(* CoDeSys 2.3.9.22 project: pr4.pro *)
(* Libraries: Util.lib 18.5.10 15:14:28, STANDARD.LIB 4.10.05 11:14:46, IECSFC.LIB 13.4.06 15:51:28, ANALYZATION.LIB 5.10.99 09:05:06 *)

(* PLC configuration (modules and I/O channels)
PLC 150 I [Root] node -1, in %IB0 out %QB0 {MinCycleLength = 1; MaxCycleLength = 5000}
  Discrete input 6 bit [ID100] node 0, in %IB0 out %QB0 {Filtrationtime = 10; Filtrationtime = 10; Filtrationtime = 10; Filtrationtime = 10; Filtrationtime = 10; Filtrationtime = 10; Visibility = No; PinCount = 6; WatchDogPeriod = 1000; PollPeriod = 1}
    AT %IX0.0 [BitInput]
    AT %IX0.1 [BitInput]
    AT %IX0.2 [BitInput]
    AT %IX0.3 [BitInput]
    AT %IX0.4 [BitInput]
    AT %IX0.5 [BitInput]
  Discrete output 4 bit [ID101] node 1, in %IB1 out %QB1 {PinCount = 4; SafeValueBool = FALSE; SafeValueBool = FALSE; SafeValueBool = FALSE; SafeValueBool = FALSE; Visibility = No}
    AT %QX1.0 [BitOutput]
    AT %QX1.1 [BitOutput]
    AT %QX1.2 [BitOutput]
    AT %QX1.3 [BitOutput]
  Special output [ID104] node 2, in %IB2 out %QB2 {Visibility = No; PinCount = 1}
    AT %QX2.0 [BitOutput] Special output
  Unifed signal sensor [ID700] node 3, in %IB3 out %QB3 {Type_of_sensor700 = IT_0_20; measure_interval = 0.8; ainlow = 0; ainhigh = 20; first_cor_point = 0; first_delta = 0; second_cor_point = 0; second_delta = 0; third_cor_point = 0; third_delta = 0; Visibility = No}
    AT %ID3.0 [FloatInput] Value
    AT %IW3.1 [WordInput] Circular time
    Analog Input [ID107] node 0, in %IB3.0 out %QB3.0
  Unifed signal sensor [ID700] node 4, in %IB4 out %QB4 {Type_of_sensor700 = IT_0_20; measure_interval = 0.8; ainlow = 0; ainhigh = 20; first_cor_point = 0; first_delta = 0; second_cor_point = 0; second_delta = 0; third_cor_point = 0; third_delta = 0; Visibility = No}
    AT %ID4.0 [FloatInput] Value
    AT %IW4.1 [WordInput] Circular time
    Analog Input [ID107] node 0, in %IB4.0 out %QB4.0
  Unifed signal sensor [ID700] node 5, in %IB5 out %QB5 {Type_of_sensor700 = IT_0_20; measure_interval = 0.8; ainlow = 0; ainhigh = 20; first_cor_point = 0; first_delta = 0; second_cor_point = 0; second_delta = 0; third_cor_point = 0; third_delta = 0; Visibility = No}
    AT %ID5.0 [FloatInput] Value
    AT %IW5.1 [WordInput] Circular time
    Analog Input [ID107] node 0, in %IB5.0 out %QB5.0
  Unifed signal sensor [ID700] node 6, in %IB6 out %QB6 {Type_of_sensor700 = IT_0_20; measure_interval = 0.8; ainlow = 0; ainhigh = 20; first_cor_point = 0; first_delta = 0; second_cor_point = 0; second_delta = 0; third_cor_point = 0; third_delta = 0; Visibility = No}
    AT %ID6.0 [FloatInput] Value
    AT %IW6.1 [WordInput] Circular time
    Analog Input [ID107] node 0, in %IB6.0 out %QB6.0
  Analog output [ID106] node 7, in %IB7 out %QB7 {DAC_Type = Current 4-20mA; Analog_offset_correction = 0; Analog_full_range_correction = 0; SafeValueFloat = 0; Visibility = No}
    AT %QD7.0 [FloatOutput] Value
  Analog output [ID106] node 8, in %IB8 out %QB8 {DAC_Type = Current 4-20mA; Analog_offset_correction = 0; Analog_full_range_correction = 0; SafeValueFloat = 0; Visibility = No}
    AT %QD8.0 [FloatOutput] Value
*)

(* POU PLC_PRG, CFC *)
PROGRAM PLC_PRG
VAR
	start: BOOL;
	pipe: BOOL;
	ctu1: CTU;
	blink1: BLINK;
	ctu2: CTU;
	wagon: REAL;
	rs1: RS;
	givePipe: BOOL;
	pipeVanish: BOOL;
	rs2: RS;
	givePipeC1: BOOL;
	givePipeC2: BOOL;
	pipeVanishC1: BOOL;
	pipeVanishC2: BOOL;
	rs3: RS;
	ctu3: CTU;
	ctu4: CTU;
	pipe1Y: REAL;
	pipe2Y: REAL;
	pipe2X: REAL;
	ctu5: CTU;
	pipe1X: REAL;
	stop: BOOL;
	loadEnd: BOOL;
	blink2: BLINK;
	wagon1: REAL;
	C1: BOOL;
	C2: BOOL;
	ctu6: CTU;
	rs4: RS;
	ctu7: CTU;
	givePipeC1ON: BOOL;
	P9: BOOL;
	ctu8: CTU;
	removePipeC1: BOOL;
	removePipeC2: BOOL;
	rs5: RS;
	ctu9: CTU;
	givePipeC2ON: BOOL;
	P0: BOOL;
	P5: BOOL;
	P6: BOOL;
	P4: BOOL;
	P3: BOOL;
	P1: BOOL;
	P2: BOOL;
	P8: BOOL;
END_VAR
VAR (* helpers for the ST form of the networks *)
	_t369 : BOOL;
	_t164 : BOOL;
	_t287 : BOOL;
	_t446 : BOOL;
	_t193 : BOOL;
	_t190 : REAL;
	_t207 : REAL;
	_t237 : REAL;
	_t321 : REAL;
	_t357 : REAL;
	_t214 : BOOL;
	_t430 : BOOL;
	_t250 : REAL;
	_t294 : REAL;
	_t315 : BOOL;
	_t445 : BOOL;
	_t241 : BOOL;
	_t231 : REAL;
	_t345 : REAL;
	_t431 : BOOL;
	_t350 : BOOL;
	_t427 : BOOL;
	_t440 : BOOL;
END_VAR
_CFC_ (* Continuous Function Chart, elements in execution order *)
#0 AND(#7.Q1, NOT #8.Q)
#1 AND(NOT stop, #16.OUT)
#2 AND(#1, #35)
#3 loadEnd <= #2
#4 AND(#7.Q1, NOT #43.Q1)
#5 S pipeVanishC1 <= NOT givePipeC1
#6 R pipeVanishC1 <= #8.Q
#7 rs2:RS(SET: givePipeC1, RESET1: #58.Q)
#8 ctu1:CTU(CU: #25, RESET: #58.Q, PV: 14)
#9 AND(#7.Q1, #1, #4)
#10 ADD(#18, #42, #51, #59, #70)
#11 wagon <= #10
#12 AND(#1, #7.Q1, NOT #27.Q)
#13 C1 <= #12
#14 AND(#24, start)
#15 rs1:RS(SET: #14, RESET1: #58.Q)
#16 blink1:BLINK(ENABLE: #15.Q1, TIMELOW: T#0.1s, TIMEHIGH: T#0.1s)
#17 WORD_TO_REAL(#8.CV)
#18 MUL(#17, -1)
#19 EQ(wagon, 0)
#20 P9 <= #19
#21 AND(#7.Q1, NOT #27.Q)
#22 givePipeC1ON <= #21
#23 EQ(pipe1Y, -44)
#24 OR(#7.Q1, #43.Q1)
#25 AND(#9, NOT #8.Q)
#26 AND(#8.Q, #9, NOT #27.Q)
#27 ctu2:CTU(CU: #26, RESET: #58.Q, PV: 22)
#28 pipe1Y <= #40
#29 AND(#39.Q, #9, NOT #30.Q)
#30 ctu6:CTU(CU: #29, RESET: #58.Q, PV: 22)
#31 MUL(#55, -1)
#32 rs4:RS(SET: #33, RESET1: #58.Q)
#33 AND(removePipeC1, #30.Q)
#34 AND(#43.Q1, #1, #74)
#35 OR(#27.Q, #45.Q)
#36 WORD_TO_REAL(#27.CV)
#37 MUL(#36, -1)
#38 AND(#27.Q, #9, NOT #39.Q)
#39 ctu3:CTU(CU: #38, RESET: #58.Q, PV: 38)
#40 ADD(#37, #47, #31, #64)
#41 WORD_TO_REAL(#39.CV)
#42 MUL(#41, -1)
#43 rs3:RS(SET: givePipeC2, RESET1: #69.Q)
#44 AND(#34, NOT #45.Q)
#45 ctu4:CTU(CU: #44, RESET: #69.Q, PV: 22)
#46 WORD_TO_REAL(#45.CV)
#47 MUL(#46, -1)
#48 AND(#45.Q, #34, NOT #49.Q)
#49 ctu5:CTU(CU: #48, RESET: #69.Q, PV: 40)
#50 WORD_TO_REAL(#49.CV)
#51 MUL(#50, -1)
#52 R pipeVanishC1 <= #43.Q1
#53 AND(#1, #43.Q1, NOT #45.Q)
#54 C2 <= #53
#55 WORD_TO_REAL(#30.CV)
#56 S pipeVanishC1 <= #32.Q1
#57 AND(#32.Q1, #9, NOT #58.Q)
#58 ctu7:CTU(CU: #57, RESET: #58.Q, PV: 52)
#59 WORD_TO_REAL(#58.CV)
#60 AND(#34, NOT #61.Q, #49.Q)
#61 ctu8:CTU(CU: #60, RESET: #69.Q, PV: 22)
#62 P1 <= #90
#63 WORD_TO_REAL(#61.CV)
#64 MUL(#63, -1)
#65 rs5:RS(SET: #66, RESET1: #69.Q)
#66 AND(removePipeC2, #61.Q)
#67 S pipeVanishC1 <= #65.Q1
#68 AND(#65.Q1, #34, NOT #69.Q)
#69 ctu9:CTU(CU: #68, RESET: #69.Q, PV: 40)
#70 WORD_TO_REAL(#69.CV)
#71 S pipeVanishC2 <= #8.Q
#72 S pipeVanishC2 <= NOT givePipeC1
#73 R pipeVanishC2 <= #0
#74 AND(#43.Q1, NOT #7.Q1)
#75 AND(#43.Q1, NOT #45.Q)
#76 givePipeC2ON <= #75
#77 EQ(wagon, -52)
#78 P0 <= #77
#79 EQ(wagon, -40)
#80 P0 <= #79
#81 EQ(wagon, -52)
#82 P5 <= #81
#83 EQ(wagon, -40)
#84 P6 <= #83
#85 EQ(pipe1Y, 0)
#86 P3 <= #91
#87 EQ(pipe1Y, 0)
#88 AND(#87, givePipeC2ON)
#89 P4 <= #88
#90 AND(#81, #23)
#91 AND(#85, givePipeC1ON)
#92 EQ(pipe1Y, -44)
#93 P2 <= #94
#94 AND(#83, #92)
#95 EQ(wagon, -14)
#96 P8 <= #95
_END_CFC_
(* the same logic as Structured Text *)
_t369 := rs2.Q1 AND NOT ctu1.Q;
_t164 := NOT stop AND blink1.OUT;
loadEnd := _t164 AND _t287;
_t446 := rs2.Q1 AND NOT rs3.Q1;
IF NOT givePipeC1 THEN pipeVanishC1 := TRUE; END_IF;
IF ctu1.Q THEN pipeVanishC1 := FALSE; END_IF;
rs2(SET := givePipeC1, RESET1 := ctu7.Q);
ctu1(CU := _t193, RESET := ctu7.Q, PV := 14);
wagon := _t190 + _t207 + _t237 + _t321 + _t357;
C1 := _t164 AND rs2.Q1 AND NOT ctu2.Q;
rs1(SET := _t214 AND start, RESET1 := ctu7.Q);
blink1(ENABLE := rs1.Q1, TIMELOW := T#0.1s, TIMEHIGH := T#0.1s);
_t190 := WORD_TO_REAL(ctu1.CV) * (-1);
P9 := wagon = 0;
givePipeC1ON := rs2.Q1 AND NOT ctu2.Q;
_t430 := pipe1Y = (-44);
_t214 := rs2.Q1 OR rs3.Q1;
_t193 := (rs2.Q1 AND _t164 AND _t446) AND NOT ctu1.Q;
ctu2(CU := ctu1.Q AND (rs2.Q1 AND _t164 AND _t446) AND NOT ctu2.Q, RESET := ctu7.Q, PV := 22);
pipe1Y := _t250;
ctu6(CU := ctu3.Q AND (rs2.Q1 AND _t164 AND _t446) AND NOT ctu6.Q, RESET := ctu7.Q, PV := 22);
rs4(SET := _t315, RESET1 := ctu7.Q);
_t315 := removePipeC1 AND ctu6.Q;
_t241 := rs3.Q1 AND _t164 AND _t445;
_t287 := ctu2.Q OR ctu4.Q;
ctu3(CU := ctu2.Q AND (rs2.Q1 AND _t164 AND _t446) AND NOT ctu3.Q, RESET := ctu7.Q, PV := 38);
_t250 := (WORD_TO_REAL(ctu2.CV) * (-1)) + _t231 + (_t294 * (-1)) + _t345;
_t207 := WORD_TO_REAL(ctu3.CV) * (-1);
rs3(SET := givePipeC2, RESET1 := ctu9.Q);
ctu4(CU := _t241 AND NOT ctu4.Q, RESET := ctu9.Q, PV := 22);
_t231 := WORD_TO_REAL(ctu4.CV) * (-1);
ctu5(CU := ctu4.Q AND _t241 AND NOT ctu5.Q, RESET := ctu9.Q, PV := 40);
_t237 := WORD_TO_REAL(ctu5.CV) * (-1);
IF rs3.Q1 THEN pipeVanishC1 := FALSE; END_IF;
C2 := _t164 AND rs3.Q1 AND NOT ctu4.Q;
_t294 := WORD_TO_REAL(ctu6.CV);
IF rs4.Q1 THEN pipeVanishC1 := TRUE; END_IF;
ctu7(CU := rs4.Q1 AND (rs2.Q1 AND _t164 AND _t446) AND NOT ctu7.Q, RESET := ctu7.Q, PV := 52);
_t321 := WORD_TO_REAL(ctu7.CV);
ctu8(CU := _t241 AND NOT ctu8.Q AND ctu5.Q, RESET := ctu9.Q, PV := 22);
P1 := _t431;
_t345 := WORD_TO_REAL(ctu8.CV) * (-1);
rs5(SET := _t350, RESET1 := ctu9.Q);
_t350 := removePipeC2 AND ctu8.Q;
IF rs5.Q1 THEN pipeVanishC1 := TRUE; END_IF;
ctu9(CU := rs5.Q1 AND _t241 AND NOT ctu9.Q, RESET := ctu9.Q, PV := 40);
_t357 := WORD_TO_REAL(ctu9.CV);
IF ctu1.Q THEN pipeVanishC2 := TRUE; END_IF;
IF NOT givePipeC1 THEN pipeVanishC2 := TRUE; END_IF;
IF _t369 THEN pipeVanishC2 := FALSE; END_IF;
_t445 := rs3.Q1 AND NOT rs2.Q1;
givePipeC2ON := rs3.Q1 AND NOT ctu4.Q;
P0 := wagon = (-52);
P0 := wagon = (-40);
P5 := wagon = (-52);
P6 := wagon = (-40);
P3 := _t427;
P4 := (pipe1Y = 0) AND givePipeC2ON;
_t431 := (wagon = (-52)) AND _t430;
_t427 := (pipe1Y = 0) AND givePipeC1ON;
P2 := _t440;
_t440 := (wagon = (-40)) AND (pipe1Y = (-44));
P8 := wagon = (-14);
END_PROGRAM

(* Visualisation viz1
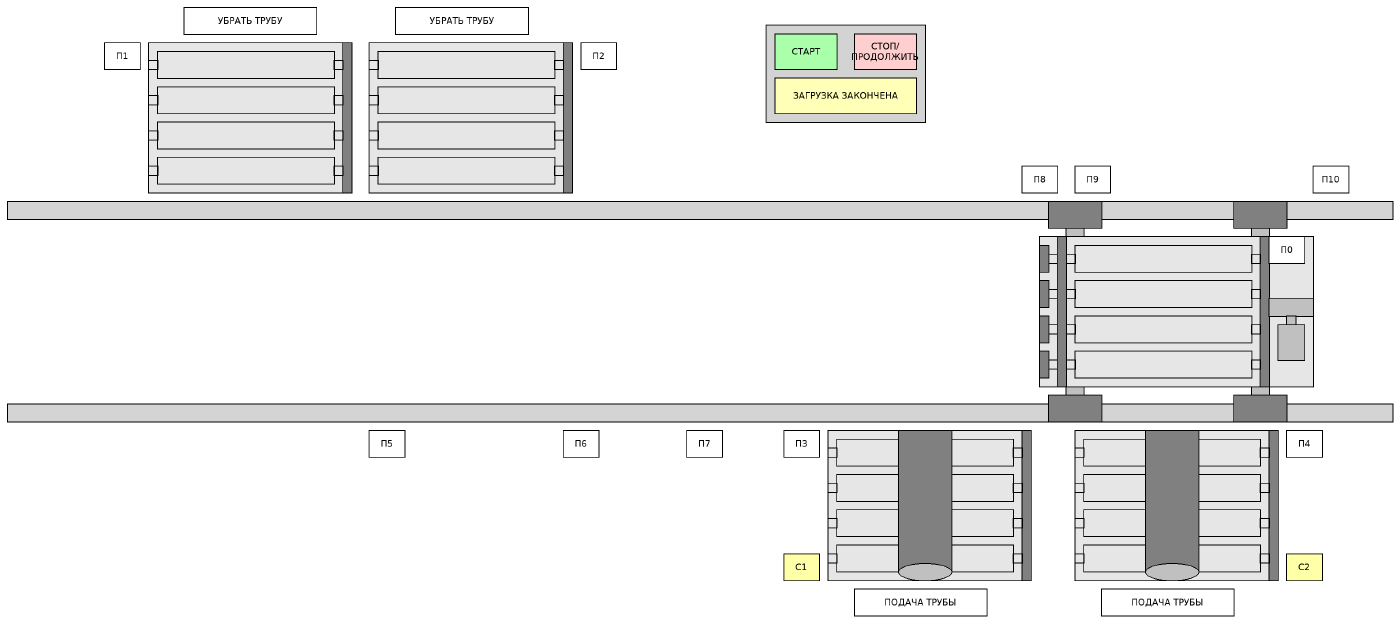
rectangle at (120,50)-(161,81): text "П1"; alarm colour if PLC_PRG.P1
rectangle at (660,50)-(701,81): text "П2"; alarm colour if PLC_PRG.P2
rectangle at (420,490)-(461,521): text "П5"; alarm colour if PLC_PRG.P5
rectangle at (640,490)-(681,521): text "П6"; alarm colour if PLC_PRG.P6
rectangle at (890,490)-(931,521): text "П3"; alarm colour if PLC_PRG.P3
rectangle at (780,490)-(821,521): text "П7"
rectangle at (1460,490)-(1501,521): text "П4"; alarm colour if PLC_PRG.P4
rectangle at (890,630)-(931,661): text "С1"; alarm colour if PLC_PRG.C1
rectangle at (1160,190)-(1201,221): text "П8"; alarm colour if PLC_PRG.P8
rectangle at (1220,190)-(1261,221): text "П9"; alarm colour if PLC_PRG.P9
rectangle at (1490,190)-(1531,221): text "П10"
group at (1180,230)-(1491,481)
  rectangle at (260,40)-(301,71): text "П0"
rounded rectangle at (880,40)-(951,81): text "СТАРТ"; alarm colour if PLC_PRG.start; taps PLC_PRG.start
rounded rectangle at (1250,670)-(1401,701): text "ПОДАЧА ТРУБЫ"; alarm colour if PLC_PRG.givePipeC2ON; taps PLC_PRG.givePipeC2
rounded rectangle at (970,670)-(1121,701): text "ПОДАЧА ТРУБЫ"; alarm colour if PLC_PRG.givePipeC1ON; taps PLC_PRG.givePipeC1
rounded rectangle at (880,90)-(1041,131): text "ЗАГРУЗКА ЗАКОНЧЕНА"; alarm colour if PLC_PRG.loadEnd
rounded rectangle at (970,40)-(1041,81): text "СТОП/ / ПРОДОЛЖИТЬ"; alarm colour if PLC_PRG.stop; toggles PLC_PRG.stop
rectangle at (1460,630)-(1501,661): text "С2"; alarm colour if PLC_PRG.C2
rounded rectangle at (210,10)-(361,41): text "УБРАТЬ ТРУБУ"; taps PLC_PRG.removePipeC1
rounded rectangle at (450,10)-(601,41): text "УБРАТЬ ТРУБУ"; taps PLC_PRG.removePipeC2
rectangle at (1440,270)-(1481,301): text "П0"; alarm colour if PLC_PRG.P0; x offset PLC_PRG.wagon*20
93 more shapes without text or variables
*)
